FUNCTION_BLOCK Basic1 (* Basic Function Block Type *)
  (* Standard: 61499-2 *)
  (* Version 0.0, 11/21/2016, chivdan, nxtControl GmbH, Template *)
  PACKAGE Main;
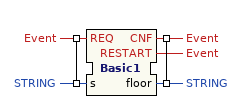
  EVENT_INPUT
    REQ WITH s; (* Normal Execution Request *)
  END_EVENT
  EVENT_OUTPUT
    CNF WITH floor; (* Execution Confirmation *)
    RESTART;
  END_EVENT
  VAR_INPUT
    s : STRING; (* Input event qualifier *)
  END_VAR
  VAR_OUTPUT
    floor : STRING; (* Output event qualifier *)
  END_VAR
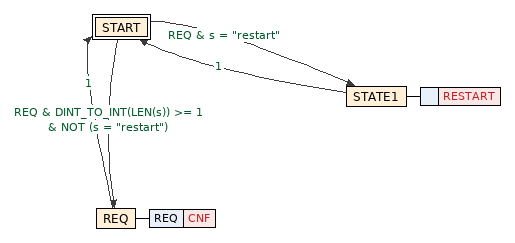
  EC_STATES
    START; (* Initial State *)
    REQ : REQ -> CNF; (* Normal execution *)
    STATE1 : -> RESTART;
  END_STATES
  EC_TRANSITIONS
    START TO REQ := REQ & DINT_TO_INT(LEN(s)) >= 1 & NOT (s = "restart");
    REQ TO START := 1;
    START TO STATE1 := REQ & s = "restart";
    STATE1 TO START := 1;
  END_TRANSITIONS
  ALGORITHM INIT IN ST: (* Initialization algorithm *)
;
  END_ALGORITHM
  ALGORITHM REQ IN ST: (* Normally executed algorithm *)
VAR
	length: INT;
	i : INT;
	tmp: STRING;
END_VAR
floor:="0";
length := DINT_TO_INT(LEN(s));
IF length = 1 THEN
	floor := s;
ELSE
  floor := MID(s, 1, 3);
END_IF;
  END_ALGORITHM
END_FUNCTION_BLOCK
